// TIA Portal V21 export
// export: Created 2026-08-26T08:41:01.564255Z, ExportSetting None, DisplayName Totally Integrated Automation Portal, DisplayVersion V21, DisplayName STEP 7 Professional, DisplayVersion V21, DisplayName STEP 7 Safety, DisplayVersion V21, DisplayName Tech WebApplication, DisplayVersion V21, DisplayName WinCC Basic/Comfort/Advanced, DisplayVersion V21
FUNCTION_BLOCK "TASK012A_NonTO_Verify"   // FB2, LAD
{ S7_Optimized_Access := 'TRUE' }
// stored: MemoryReserve 100, SetENOAutomatically false
   VAR_INPUT
      Start : Bool;
      Stop : Bool;
      CountPulse : Bool;
      CountReset : Bool;
      PresetValue : Int;
      DelayIn : Bool;
      FallIn : Bool;
      FcEnable : Bool;
      FbEnable : Bool;
   END_VAR
   VAR_OUTPUT
      Motor : Bool;
      CountDone : Bool;
      CountValue : Int;
      TofQ : Bool;
      FallPulse : Bool;
      FcOk : Bool;
      FbActive : Bool;
   END_VAR
   VAR
      OffDelay { S7_SetPoint := 'True'} : TOF_TIME;
      BatchCnt { S7_SetPoint := 'True'} : CTU_INT;
      FallMem : Bool;
      Child { S7_SetPoint := 'True'} : "TASK012A_FB_Callee";
   END_VAR
   VAR_TEMP   // added for the SCL form of the ladder/FBD networks
      _w1 : Bool;
   END_VAR
BEGIN

REGION Network 1
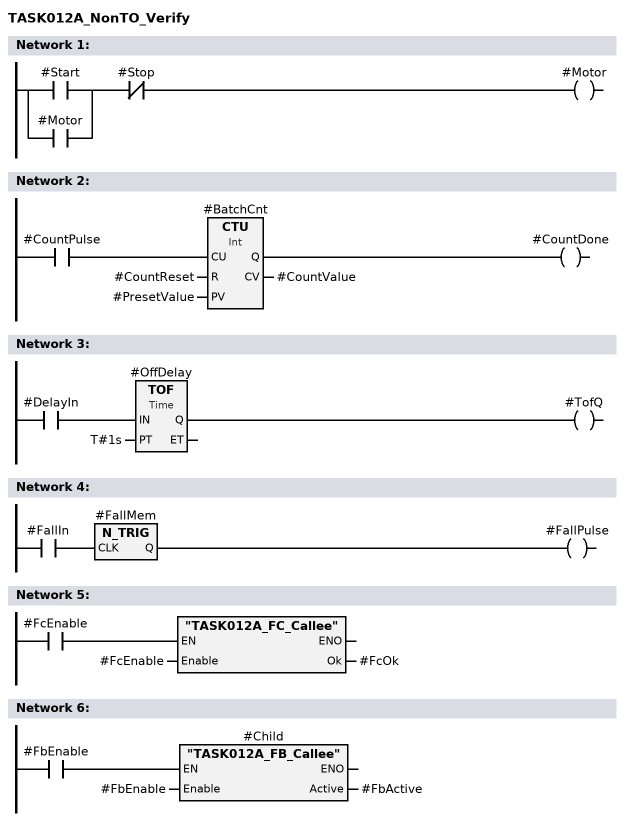
   RUNG wire#powerrail
      Contact( #Start )
      wire#w1
      I_Contact( #Stop )
      Coil( #Motor )
   END_RUNG
   RUNG wire#powerrail
      Contact( #Motor )
   END_RUNG wire#w1
   // the same network as SCL:
   #Motor := (#Start OR #Motor) AND NOT #Stop;
END_REGION

REGION Network 2
   RUNG wire#powerrail
      Contact( #CountPulse )
      { S7_Templates := "value_type := Int" } #BatchCnt.CTU(r := #CountReset, pv := #PresetValue, cv => #CountValue)
      Coil( #CountDone )
   END_RUNG
   // the same network as SCL:
   #BatchCnt(CU := #CountPulse, R := #CountReset, PV := #PresetValue, CV => #CountValue);   // CTU
   #CountDone := #BatchCnt.Q;
END_REGION

REGION Network 3
   RUNG wire#powerrail
      Contact( #DelayIn )
      { S7_Templates := "time_type := Time" } #OffDelay.TOF(pt := T#1s, et =>)
      Coil( #TofQ )
   END_RUNG
   // the same network as SCL:
   #OffDelay(IN := #DelayIn, PT := T#1s);   // TOF
   #TofQ := #OffDelay.Q;
END_REGION

REGION Network 4
   RUNG wire#powerrail
      Contact( #FallIn )
      N_Trig( #FallMem )
      Coil( #FallPulse )
   END_RUNG
   // the same network as SCL:
   #_w1 := NOT #FallIn AND #FallMem;   // falling edge
   #FallMem := #FallIn;
   #FallPulse := #_w1;
END_REGION

REGION Network 5
   RUNG wire#powerrail
      Contact( #FcEnable )
      "TASK012A_FC_Callee"(Enable := #FcEnable, Ok => #FcOk)
   END_RUNG
   // the same network as SCL:
   IF #FcEnable THEN "TASK012A_FC_Callee"(Enable := #FcEnable, Ok => #FcOk); END_IF;
END_REGION

REGION Network 6
   RUNG wire#powerrail
      Contact( #FbEnable )
      #Child(Enable := #FbEnable, Active => #FbActive)
   END_RUNG
   // the same network as SCL:
   IF #FbEnable THEN
       #Child(Enable := #FbEnable, Active => #FbActive);   // "TASK012A_FB_Callee"
   END_IF;
END_REGION
END_FUNCTION_BLOCK
